FUNCTION_BLOCK Skill_Greifer_Pos_Anfahren	IMPLEMENTS I_Skill_SmartGreifer
VAR_INPUT
	// Zu verwendetes Objekt
	Objekt						:I_Objekt_SmartGreifer;	
	
	// Betriebsvariablen 
	eSysCommand					:eSystemCommand; 						// Systembefehl an Skill
	eSysState					:eSystemState;							// Momentaner Zustand des Systems
END_VAR
VAR_OUTPUT
	iErrorID					:INT;									// Fehlercode für System
END_VAR
VAR
	// Managementvariablen
	iState				:eSkillState;									// Information über Zustand von Skill
	SendDelay			:TON;
	
	// Managementvariablen 
	bGestartet			:BOOL;
	bGestoppt			:BOOL;
	
	// Zustandsvariablen
	bStarten			:BOOL;
	bStoppen			:BOOL;
	bObjektFertig		:BOOL;
	bWertErreicht		:BOOL;				
	bLimitErreicht		:BOOL;				
	bSkillFertig		:BOOL;
	bFehler				:BOOL;
	bResetten			:BOOL;
	
	// Prozessparameter
	eGreiferParam	 			:sSmartGreiferProzessVariablen;
	eGreiferParamReset			:sSmartGreiferProzessVariablen;

	ParamArray					:ARRAY[0..10] OF sSmartGreiferProzessVariablen;
	Counter						:INT;
END_VAR

// Instanzierung
SendDelay(PT := T#2ms);

// Fehlerüberwachung
IF bFehler THEN
	iState := 3;
END_IF

//_______________________________________________________________
// Reaktion auf Input-Variablen:
	// Stoppen
	IF eSysCommand = 3 THEN
		bStoppen := M_Stop();
	ELSE 
		bStoppen := FALSE;
	END_IF

	// Resetten 
	IF eSysCommand = 4 THEN
		bResetten := M_Reset();
	ELSE
		bResetten := FALSE;
	END_IF
//_______________________________________________________________
// Zustandsmanagement
CASE iState OF 
0: 	// BEREIT	
		// DO
		IF Objekt.P_State = 3 THEN		// Objekt wurde eingeschalten
			bStarten := TRUE;
		END_IF
		
		// TRANSITION
		IF bStarten	 THEN		
			bStarten := FALSE;
			iState := 1;	
		END_IF
		
		
// _________________________________________________________________________________________________________________________
1: 	// LAUFEND
		// DO			
			// Stoppen durch Sysezm
			IF bStoppen THEN																								// Transition wenn System das Orbjekt stoppt
				bGestoppt := TRUE;
			END_IF
			
			// Objekt hat sich selber gestoppt
			IF Objekt.P_State = 4 THEN																							// Objekt hat Prozess abgeschlossen
				bObjektFertig := TRUE;																							// Objekt ist fertig und wieder bereit
			END_IF
			
		// TRANSITION 
		IF bGestoppt THEN																								// Transition zu BEREIT
			bGestoppt := FALSE;																				
			iState := 0;
		END_IF
		
		IF bObjektFertig THEN																							// Transition zu ABGESCHLOSSEN
			bObjektFertig := FALSE;																							// Skill wird nicht mehr ausgeführt
			iState := 2;																									// Objekt ist fertig und wieder bereit
		END_IF
		
		IF bLimitErreicht AND Objekt.P_State = 5 THEN																							// Transition zu LIMIT
			iState := 4;
		END_IF
		
		IF bWertErreicht AND Objekt.P_State = 5 THEN																							// Transition zu ERREICHT
			iState := 5;
		END_IF
			
// _________________________________________________________________________________________________________________________			
2: 	// ABGESCHLOSSEN
		// DO
		M_Reset();
		 
		IF Objekt.P_State = 1 THEN																							// Objekt wurde geresettet
			bSkillFertig := TRUE;									
		END_IF
			
		//  TRANSITION
		IF bSkillFertig THEN
			bSkillFertig := FALSE;																																											// Resetten von Objekt
			iState := 0;
		END_IF
		
// _________________________________________________________________________________________________________________________
3: 	// FEHLER
		// DO 	
		
		// TRANSITION
		IF bResetten THEN
			iState := 0;
		END_IF
		
END_CASE

METHOD M_Reset : BOOL
Objekt.M_Reset();
eGreiferParam := eGreiferParamReset;
END_METHOD

METHOD M_Start : BOOL
// Prüfen von Bedingungen
	// Ist das  System im korrekten Status
	IF eSysState = 1 THEN
		// Ist der Skill im korrekten Status 
		IF iState = 0 THEN
			// Prüfen auf Fehler (Muss ergänzt werden)
				SendDelay(IN := TRUE);
					
				IF SendDelay.Q THEN
					Objekt.P_Prozessparameter := eGreiferParam;
					Objekt.M_Start();
					SendDelay(IN := FALSE);
					
					
					ParamArray[Counter] := eGreiferParam;
					Counter := Counter + 1;
				END_IF
					
		END_IF
	END_IF
END_METHOD

METHOD M_Stop : BOOL
Objekt.M_Stop();
eGreiferParam := eGreiferParamReset;
END_METHOD

PROPERTY P_SGripperParam : sSmartGreiferProzessVariablen
SET
eGreiferParam := P_SGripperParam;
END_SET
END_PROPERTY

PROPERTY P_State : eSkillState
GET
P_State := iState;
END_GET
END_PROPERTY

END_FUNCTION_BLOCK

(* stored: Version 1.1.0.1
   POU Skill_Greifer_Pos_Anfahren: Id {98210e8f-b577-460a-824e-a40bbe292bb9}, SpecialFunc None
   Folder 01_Steuerungsmethoden: Id {ce4f4fae-0d80-421d-ad11-2f1af775784f}
   Folder 02_Steuerungseigenschaften: Id {9bc7b88e-6bad-4969-9dcc-a138a59804b7}
   Folder 03_Prozesseigenschaften: Id {f245a847-91cc-4c3b-ae26-c2f97efdc277}
   Method M_Reset: Id {9681675d-c826-49e1-9762-1d6a3b1f0fd3}
   Method M_Start: Id {adfcfbf0-fd5e-42b6-8ae7-e20aed73ac37}
   Method M_Stop: Id {fa3fe864-0fc2-487f-b91b-4465f36ebd46}
   Property P_SGripperParam: Id {24a56df2-d061-4605-a850-faa49bdd332b}
   Set Set: Id {94fe09d4-c7e2-4360-93ce-cdf0ae2858fd}
   Property P_State: Id {0f0ba2d7-8962-499e-bf02-77f7f3aa889f}
   Get Get: Id {77be5290-7de1-4b4e-a3f0-fb8b4aa0a089} *)
